FUNCTION_BLOCK Resource3nm
  (* Version 1.0, 2008-12-16, Goran Cengic, Chalmers *)
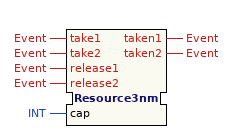
  EVENT_INPUT
    take1;
    take2;
    release1;
    release2;
  END_EVENT
  EVENT_OUTPUT
    taken1;
    taken2;
  END_EVENT
  VAR_INPUT
    cap : INT;
  END_VAR
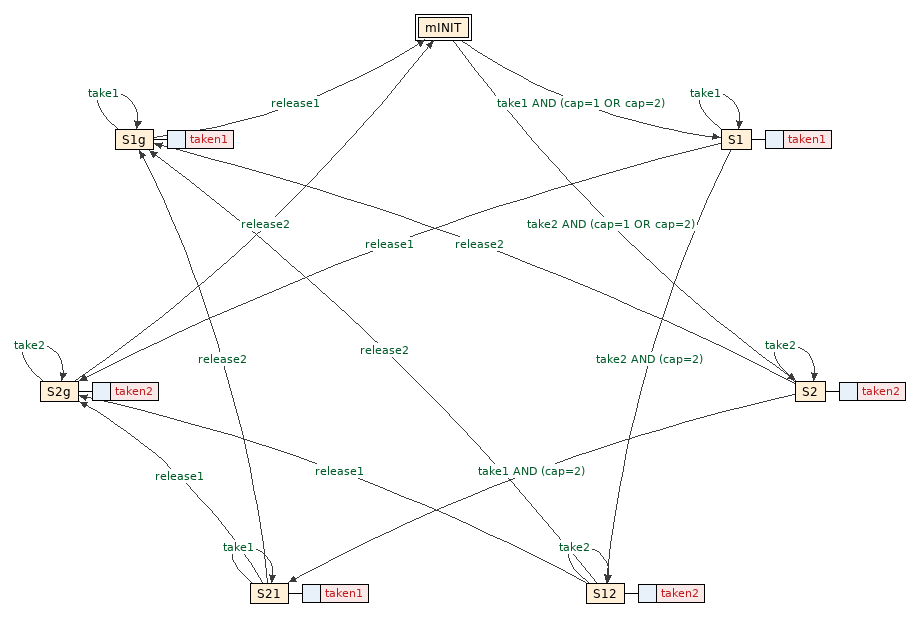
  EC_STATES
    mINIT;
    S1 : -> taken1;
    S2 : -> taken2;
    S12 : -> taken2;
    S21 : -> taken1;
    S2g : -> taken2;
    S1g : -> taken1;
  END_STATES
  EC_TRANSITIONS
    mINIT TO S1 := take1 AND (cap=1 OR cap=2);
    S1 TO S1 := take1;
    S1 TO S2g := release1;
    S2g TO S2g := take2;
    S2g TO mINIT := release2;
    mINIT TO S2 := take2 AND (cap=1 OR cap=2);
    S2 TO S2 := take2;
    S2 TO S1g := release2;
    S1g TO S1g := take1;
    S1g TO mINIT := release1;
    S1 TO S12 := take2 AND (cap=2);
    S12 TO S12 := take2;
    S12 TO S2g := release1;
    S12 TO S1g := release2;
    S2 TO S21 := take1 AND (cap=2);
    S21 TO S21 := take1;
    S21 TO S1g := release2;
    S21 TO S2g := release1;
  END_TRANSITIONS
END_FUNCTION_BLOCK
